TYPE Interval :
STRUCT
	startPos : REAL;
	endPos : REAL;
END_STRUCT
END_TYPE

(* stored: Version 1.1.0.1, ProductVersion 3.1.4024.11
   DUT Interval: Id {f20c923f-8b47-4de8-9987-10b904ebc0dc} *)
